FUNCTION_BLOCK TIME_Param
VAR_INPUT PERSISTENT
	val			: TIME;
END_VAR

END_FUNCTION_BLOCK

(* stored: Version 1.1.0.1
   POU TIME_Param: Id {b9e690dc-3b3c-4b20-9d56-258bd76f5a4c}, SpecialFunc None *)
